// TIA Portal V20 export
TYPE "LER_typeCommunicationBRCVMonitoring"
// stored: Access Published
   STRUCT
      len : Word;
      ndr : Bool := false;
      error : Bool := false;
      status : Word := 16#0;
   END_STRUCT;
END_TYPE
